{attribute 'qualified_only'}
{attribute 'strict'}
TYPE MC_StartMode :
(
	mcAbsolute := 0,
	mcRelative := 1,
	mcRampIn := 2
);
END_TYPE

(* stored: Version 1.1.0.1, ProductVersion 3.1.4024.11
   DUT MC_StartMode: Id {828a79e6-719c-4255-b105-b022203c39d0} *)
